FUNCTION_BLOCK abstract FB_FlyingBase
VAR
  _eCheck               : E_CHECK_STATE;
  _bError               : BOOL;
  _nErrorId             : UDINT;

  _ItfAxis              : I_McAxis;               // slave to the rythm.
  _Master               : REFERENCE TO AXIS_REF;  // obey I must

  _rModulo              : LREAL;                  // modulo length/angle of NC axis.

  _stFlyData            : ST_FLY_DATA;
  _stMoveData           : ST_AXIS_MOVE_DATA;
  _stOptions            : ST_FLY_OPTIONS;

  _szSyncMode           : ARRAY[1..2] OF UINT;
  _stSyncMode           : Tc2_MC2_FlyingSaw.ST_SyncMode;
  _stGearInPosOptions   : Tc2_MC2_FlyingSaw.ST_GearInPosOptions;
  _stGearInVeloOptions  : Tc2_MC2_FlyingSaw.ST_GearInVeloOptions;

  _fbGearInPos          : Tc2_MC2_FlyingSaw.MC_GearInPos;   // position based gearing
  _fbGearInVelo         : Tc2_MC2_FlyingSaw.MC_GearInVelo;  // velocity based gearing
  //_fbReadCharacter      : Tc2_MC2_FlyingSaw.MC_ReadFlyingSawCharacteristics; 

  _MessageLevel         : E_MessageType;
  _stMsg                : ST_Message;
END_VAR

PROPERTY AxisModulo : lreal
SET
_rModulo := AxisModulo;
END_SET
END_PROPERTY

METHOD GearInPos : E_PROGRESS
VAR_INPUT
  Execute             : BOOL;
  stMoveData          : ST_AXIS_MOVE_DATA;
  stGearData          : ST_FLY_DATA;
  stOptions           : ST_FLY_OPTIONS; 
END_VAR
VAR_INST
  _nErrorId           : UDINT;
  _rPosLate,
  _rPos               : LREAL;
  _eState             : E_PROGRESS;
END_VAR
IF NOT Execute THEN _eState       := E_PROGRESS.PROGRESS_INIT; END_IF
 
IF NOT (_ItfAxis <> 0)         THEN GearInPos    := E_PROGRESS.PROGRESS_ERROR; RETURN; END_IF


CASE _eState
OF
  E_PROGRESS.PROGRESS_INIT:
    IF Execute
    THEN
      _bError                 := FALSE;
      _rPosLate               := 0.0;
      _nErrorId               := 0;
      _eState                 := E_PROGRESS.PROGRESS_BUSY;

      _stGearInPosOptions.PositionLimitMin  := stOptions.PositionLimitMin;
      _stGearInPosOptions.PositionLimitMax  := stOptions.PositionLimitMax;

      memcpy(ADR(_stSyncMode), ADR(stOptions.SyncMode), SIZEOF(_stSyncMode));

      IF NOT __ISVALIDREF(_Master)
      THEN
        _bError               := TRUE;
        _nErrorId             := 666;
        _eState               := E_PROGRESS.PROGRESS_ERROR;

        _stMsg.eType          := E_MessageType.eMessageError;
        _stMsg.eSubdevice     := e_Subdevice.fbGearInPos;
        _stMsg.iErrorNumber   := _nErrorId;
        _stMsg.sText          := concat('Invalid Master Ref: ', TO_STRING(_eState));
        f_MessageSet(_stMsg);

      ELSIF (_ItfAxis.AxisRef.NcToPlc.ModuloActPos > stGearData.rModuloSyncPosSlave + stGearData.rDelta)
      THEN
        _bError               := TRUE;
        _rPosLate             := _ItfAxis.AxisRef.NcToPlc.ModuloActPos;
        _rPos                 := stGearData.rModuloSyncPosSlave + stGearData.rDelta;

        _nErrorId             := 667;
        _eState               := E_PROGRESS.PROGRESS_ERROR;

        _stMsg.eType          := E_MessageType.eMessageError;
        _stMsg.eSubdevice     := e_Subdevice.fbGearInPos;
        _stMsg.iErrorNumber   := _nErrorId;
        _stMsg.sText          := concat('ModuloActPos: ', TO_STRING(_rPosLate));
        _stMsg.sText          := concat(_stMsg.sText, '; ModuloSyncPosSlave + stGearData.rDelta: ');
        _stMsg.sText          := concat(_stMsg.sText, TO_STRING(_rPos));
        f_MessageSet(_stMsg);
      END_IF
    END_IF
END_CASE
//-----------------------------------------------------------------------------
//-----------------------------------------------------------------------------
CASE _eState
OF
  E_PROGRESS.PROGRESS_BUSY:
    _eState                   := E_PROGRESS.PROGRESS_PREPARE;

    _fbGearInPos(
        Master                := _Master, 
        Slave                 := _ItfAxis.AxisRef, 
        Execute               := FALSE, 

        RatioNumerator        := stGearData.rGearNumerator, 
        RatioDenominator      := stGearData.iGearDenumerator, 

        MasterSyncPosition    := _Master.NcToPlc.ActPos 
                               + stGearData.rDeltaToMasterPos,                            // absolute position

        SlaveSyncPosition     := ABS(_ItfAxis.AxisRef.NcToPlc.ModuloActTurns)*_rModulo
                               + stGearData.rModuloSyncPosSlave,                          // absolute position

        SyncMode              := _stSyncMode,
        MasterStartDistance   := stGearData.rMasterStartDistance,                         // if <> 0 --> master has to move before this fb does anything
        Velocity              := stMoveData.rSetVelo, 
        Acceleration          := stMoveData.rAcc, 
        Deceleration          := stMoveData.rAcc, 
        Jerk                  := stMoveData.rJerk, 
        BufferMode            := Tc2_MC2.MC_BufferMode.MC_Aborting, 
        Options               := _stGearInPosOptions, 
        ErrorID               => _nErrorId);

        IF (_MessageLevel = E_MessageType.eMessageVerbose)
        THEN
          _stMsg.eType        := E_MessageType.eMessageVerbose;
          _stMsg.eSubdevice   := e_Subdevice.fbGearInPos;
          _stMsg.iErrorNumber := _nErrorId;
          _stMsg.sText        := TO_STRING(_eState);
          f_MessageSet(_stMsg);
        END_IF
END_CASE
//-----------------------------------------------------------------------------
//-----------------------------------------------------------------------------
CASE _eState
OF
  E_PROGRESS.PROGRESS_PREPARE:
    _fbGearInPos(
        Master                := _Master, 
        Slave                 := _ItfAxis.AxisRef, 
        Execute               := TRUE);

    IF _fbGearInPos.Error
    THEN
      _bError                 := TRUE;
      _nErrorId               := _fbGearInPos.ErrorId;

      _fbGearInPos(
        Master                := _Master, 
        Slave                 := _ItfAxis.AxisRef, 
        Execute               := FALSE);

      _eState                 := E_PROGRESS.PROGRESS_ERROR;

      _stMsg.eType            := E_MessageType.eMessageError;
      _stMsg.eSubdevice       := e_Subdevice.fbGearInPos;
      _stMsg.iErrorNumber     := _nErrorId;
      _stMsg.sText            := TO_STRING(_eState);
      f_MessageSet(_stMsg);

    ELSIF _fbGearInPos.CommandAborted
    THEN
      _bError                 := TRUE;
      _eState                 := E_PROGRESS.PROGRESS_OCCUPIED;

      _stMsg.eType            := E_MessageType.eMessageWarning;
      _stMsg.eSubdevice       := e_Subdevice.fbGearInPos;
      _stMsg.iErrorNumber     := _nErrorId;
      _stMsg.sText            := concat(TO_STRING(_eState), ': CommandAborted');
      f_MessageSet(_stMsg);

      _fbGearInPos(
        Master                := _Master, 
        Slave                 := _ItfAxis.AxisRef, 
        Execute               := FALSE);

    ELSIF _fbGearInPos.InSync
    THEN
      _eState                 := E_PROGRESS.PROGRESS_DONE;

      IF (_MessageLevel > E_MessageType.eMessageError)
      THEN
        _stMsg.eType          := E_MessageType.eMessageInfo;
        _stMsg.eSubdevice     := e_Subdevice.fbGearInPos;
        _stMsg.iErrorNumber   := _nErrorId;
        _stMsg.sText          := TO_STRING(_eState);
        f_MessageSet(_stMsg);
      END_IF
      _fbGearInPos(
        Master                := _Master, 
        Slave                 := _ItfAxis.AxisRef, 
        Execute               := FALSE);
    END_IF
END_CASE
//-----------------------------------------------------------------------------
//-----------------------------------------------------------------------------
GearInPos                     := _eState;
END_METHOD

METHOD GearInVelo : E_PROGRESS
VAR_INPUT
  Execute             : BOOL;
  stMoveData          : ST_AXIS_MOVE_DATA;
  stGearData          : ST_FLY_DATA;
  stOptions           : ST_FLY_OPTIONS; 
END_VAR
VAR_INST
  _nErrorId           : UDINT;
  _rPosLate,
  _rPos               : LREAL;
  _eState             : E_PROGRESS;
END_VAR
IF NOT Execute THEN _eState       := E_PROGRESS.PROGRESS_INIT; END_IF
 
IF NOT (_ItfAxis <> 0)         THEN GearInVelo    := E_PROGRESS.PROGRESS_ERROR; RETURN; END_IF


CASE _eState
OF
  E_PROGRESS.PROGRESS_INIT:
    IF Execute
    THEN
      _nErrorId               := 0;
      _eState                 := E_PROGRESS.PROGRESS_BUSY;

      _stGearInVeloOptions.PositionLimitMin := stOptions.PositionLimitMin;
      _stGearInVeloOptions.PositionLimitMax := stOptions.PositionLimitMax;

      memcpy(ADR(_stSyncMode), ADR(stOptions.SyncMode), SIZEOF(_stSyncMode));

      IF NOT __ISVALIDREF(_Master)
      THEN
        _bError               := TRUE;
        _nErrorId             := 666;
        _eState               := E_PROGRESS.PROGRESS_ERROR;

        _stMsg.eType          := E_MessageType.eMessageError;
        _stMsg.eSubdevice     := e_Subdevice.fbGearInVelo;
        _stMsg.iErrorNumber   := _nErrorId;
        _stMsg.sText          := concat('Invalid Master Ref: ', TO_STRING(_eState));
        f_MessageSet(_stMsg);
      END_IF
    END_IF
END_CASE
//-----------------------------------------------------------------------------
//-----------------------------------------------------------------------------
CASE _eState
OF
  E_PROGRESS.PROGRESS_BUSY:
    _eState                   := E_PROGRESS.PROGRESS_PREPARE;

    _fbGearInVelo(
        Master                := _Master, 
        Slave                 := _ItfAxis.AxisRef, 
        Execute               := FALSE, 

        RatioNumerator        := stGearData.rGearNumerator, 
        RatioDenominator      := stGearData.iGearDenumerator, 

	      SyncMode:= , 
        Velocity              := stMoveData.rSetVelo, 
        Acceleration          := stMoveData.rAcc, 
        Deceleration          := stMoveData.rAcc, 
        Jerk                  := stMoveData.rJerk, 
        BufferMode            := Tc2_MC2.MC_BufferMode.MC_Aborting, 
        Options               := _stGearInVeloOptions, 
        ErrorID               => _nErrorId);

        IF (_MessageLevel = E_MessageType.eMessageVerbose)
        THEN
          _stMsg.eType        := E_MessageType.eMessageVerbose;
          _stMsg.eSubdevice   := e_Subdevice.fbGearInVelo;
          _stMsg.iErrorNumber := _nErrorId;
          _stMsg.sText        := TO_STRING(_eState);
          f_MessageSet(_stMsg);
        END_IF
END_CASE
//-----------------------------------------------------------------------------
//-----------------------------------------------------------------------------
CASE _eState
OF
  E_PROGRESS.PROGRESS_PREPARE:
    _fbGearInVelo(
        Master                := _Master, 
        Slave                 := _ItfAxis.AxisRef, 
        Execute               := TRUE);

    IF _fbGearInVelo.Error
    THEN
      _bError                 := TRUE;
      _nErrorId               := _fbGearInVelo.ErrorId;

      _fbGearInVelo(
        Master                := _Master, 
        Slave                 := _ItfAxis.AxisRef, 
        Execute               := FALSE);

      _eState                 := E_PROGRESS.PROGRESS_ERROR;

      _stMsg.eType            := E_MessageType.eMessageError;
      _stMsg.eSubdevice       := e_Subdevice.fbGearInVelo;
      _stMsg.iErrorNumber     := _nErrorId;
      _stMsg.sText            := TO_STRING(_eState);
      f_MessageSet(_stMsg);

    ELSIF _fbGearInVelo.CommandAborted
    THEN
      _bError                 := TRUE;
      _eState                 := E_PROGRESS.PROGRESS_OCCUPIED;

      _stMsg.eType            := E_MessageType.eMessageWarning;
      _stMsg.eSubdevice       := e_Subdevice.fbGearInVelo;
      _stMsg.iErrorNumber     := _nErrorId;
      _stMsg.sText            := concat(TO_STRING(_eState), ': CommandAborted');
      f_MessageSet(_stMsg);

    ELSIF _fbGearInVelo.InSync
    THEN
      _eState                 := E_PROGRESS.PROGRESS_DONE;

      IF (_MessageLevel > E_MessageType.eMessageError)
      THEN
        _stMsg.eType          := E_MessageType.eMessageInfo;
        _stMsg.eSubdevice     := e_Subdevice.fbGearInVelo;
        _stMsg.iErrorNumber   := _nErrorId;
        _stMsg.sText          := TO_STRING(_eState);
        f_MessageSet(_stMsg);
      END_IF
      _fbGearInVelo(
        Master                := _Master, 
        Slave                 := _ItfAxis.AxisRef, 
        Execute               := FALSE);
    END_IF
END_CASE
//-----------------------------------------------------------------------------
//-----------------------------------------------------------------------------
GearInVelo                    := _eState;
END_METHOD

PROPERTY MessageLevel : E_MessageType
SET
_MessageLevel := MessageLevel;
END_SET
END_PROPERTY

END_FUNCTION_BLOCK

(* stored: Version 1.1.0.1, ProductVersion 3.1.4026.19
   POU FB_FlyingBase: Id {86dcc0cc-c619-4cf3-a8fb-dd8062daa261}, SpecialFunc None
   Folder methods: Id {608bed0b-32e7-45ae-8191-54ea3d9b989c}
   Folder properties: Id {d01f30b3-daa9-4973-8211-b87183d3fae6}
   Property AxisModulo: Id {fa7d2e7f-df3c-49d5-bc43-a5ffce6c775d}
   Set Set: Id {19581ea4-e32b-45a7-871e-18a7b24dbfaf}
   Method GearInPos: Id {1420a175-40e0-489e-92fe-2ab56883c746}
   Method GearInVelo: Id {7d3d5e9c-869e-4d6e-a371-b333882c434f}
   Property MessageLevel: Id {08d2ea8c-5238-4fc8-ae70-3c4e99f8afc7}
   Set Set: Id {beca9d4b-a8c0-46e8-89fb-759253069974} *)
